{attribute 'qualified_only'}
VAR_GLOBAL
	CalculationEventClass: INT;
END_VAR

(* stored: Version 1.1.0.1, ProductVersion 3.1.4022.18
   GVL GVL: Id {c0e54612-2934-472d-898a-8f56423e9b6c} *)
